% RSLogix 500 project Práctica 3.RSS, saved by version 8.30.00.16 %
PROJECT "UNTITLED"    % processor: Bul.1763 MicroLogix 1100 Series B %

PROGRAM FILES
  LAD 2   12 rungs

DATA FILES
  O0 OUTPUT  4 elements
  I1 INPUT  6 elements
  S2 STATUS  66 elements
  B3 BINARY  1 elements
  T4 TIMER  1 elements
  C5 COUNTER  1 elements
  R6 CONTROL  1 elements
  N7 INTEGER  1 elements
  F8 FLOAT  1 elements

LADDER 2
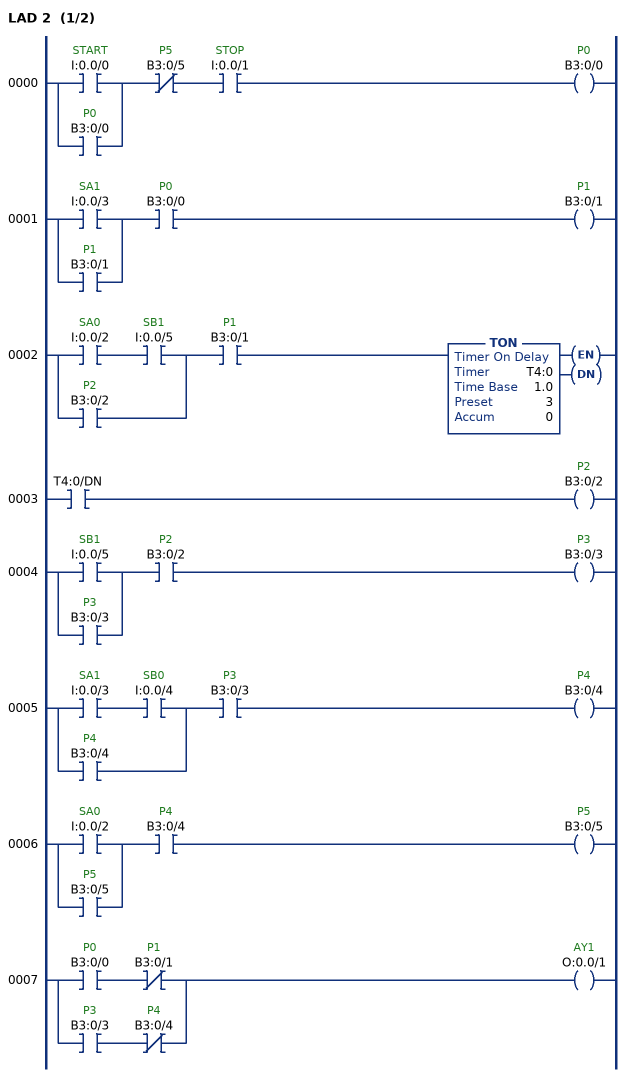
% Rung: 0 %
SOR BST XIC I:0.0/0 NXB XIC B3:0/0 BND XIO B3:0/5 XIC I:0.0/1 OTE B3:0/0 EOR
%   I:0.0/0  START %
%   B3:0/0  P0 %
%   B3:0/5  P5 %
%   I:0.0/1  STOP %
% Rung: 1 %
SOR BST XIC I:0.0/3 NXB XIC B3:0/1 BND XIC B3:0/0 OTE B3:0/1 EOR
%   I:0.0/3  SA1 %
%   B3:0/1  P1 %
%   B3:0/0  P0 %
% Rung: 2 %
SOR BST XIC I:0.0/2 XIC I:0.0/5 NXB XIC B3:0/2 BND XIC B3:0/1 TON T4:0 1.0 3 0 EOR
%   I:0.0/2  SA0 %
%   I:0.0/5  SB1 %
%   B3:0/2  P2 %
%   B3:0/1  P1 %
% Rung: 3 %
SOR XIC T4:0/DN OTE B3:0/2 EOR
%   B3:0/2  P2 %
% Rung: 4 %
SOR BST XIC I:0.0/5 NXB XIC B3:0/3 BND XIC B3:0/2 OTE B3:0/3 EOR
%   I:0.0/5  SB1 %
%   B3:0/3  P3 %
%   B3:0/2  P2 %
% Rung: 5 %
SOR BST XIC I:0.0/3 XIC I:0.0/4 NXB XIC B3:0/4 BND XIC B3:0/3 OTE B3:0/4 EOR
%   I:0.0/3  SA1 %
%   I:0.0/4  SB0 %
%   B3:0/4  P4 %
%   B3:0/3  P3 %
% Rung: 6 %
SOR BST XIC I:0.0/2 NXB XIC B3:0/5 BND XIC B3:0/4 OTE B3:0/5 EOR
%   I:0.0/2  SA0 %
%   B3:0/5  P5 %
%   B3:0/4  P4 %
% Rung: 7 %
SOR BST XIC B3:0/0 XIO B3:0/1 NXB XIC B3:0/3 XIO B3:0/4 BND OTE O:0.0/1 EOR
%   B3:0/0  P0 %
%   B3:0/1  P1 %
%   B3:0/3  P3 %
%   B3:0/4  P4 %
%   O:0.0/1  AY1 %

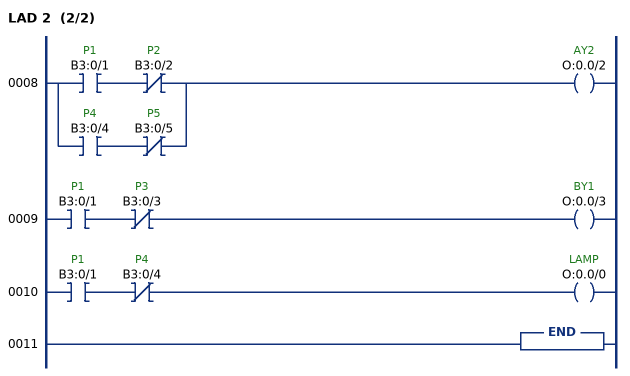
% Rung: 8 %
SOR BST XIC B3:0/1 XIO B3:0/2 NXB XIC B3:0/4 XIO B3:0/5 BND OTE O:0.0/2 EOR
%   B3:0/1  P1 %
%   B3:0/2  P2 %
%   B3:0/4  P4 %
%   B3:0/5  P5 %
%   O:0.0/2  AY2 %
% Rung: 9 %
SOR XIC B3:0/1 XIO B3:0/3 OTE O:0.0/3 EOR
%   B3:0/1  P1 %
%   B3:0/3  P3 %
%   O:0.0/3  BY1 %
% Rung: 10 %
SOR XIC B3:0/1 XIO B3:0/4 OTE O:0.0/0 EOR
%   B3:0/1  P1 %
%   B3:0/4  P4 %
%   O:0.0/0  LAMP %
% Rung: 11 %
SOR END EOR

DATA TABLE (non-zero values as saved)
DATA T4
% .PRE .ACC %
% T4:0 % 3 0
